TYPE "ModeGenStruct"
VERSION : 0.1
   STRUCT
      Out : "ModeOutStruct";
   END_STRUCT;

END_TYPE

